FUNCTION_BLOCK FB_Sequence IMPLEMENTS I_Sequence
VAR_INPUT
END_VAR
VAR_OUTPUT
	nNumber:				INT;
END_VAR
VAR
	bStarted:				Bool;
END_VAR

// Quite a lot to do here :-(

METHOD PUBLIC M_Await 
VAR_INPUT
	Message:				STRING(255);
	tTimeout:				TIME;
	bCondition:				BOOL;
	nNumber:				INT;
END_VAR
IF bStarted THEN
	IF bCondition THEN
		THIS^.nNumber:= nNumber;
	END_IF
END_IF
END_METHOD

METHOD M_Reset : BOOL
M_Stop();
nNumber:= -32768;
END_METHOD

METHOD M_Start
bStarted:= TRUE;
END_METHOD

METHOD M_Stop : BOOL
bStarted:= FALSE;
END_METHOD

PROPERTY PUBLIC P_Number : int
GET
P_Number:= nNumber;
END_GET
SET
nNumber:= P_Number;
END_SET
END_PROPERTY

END_FUNCTION_BLOCK

(* stored: Version 1.1.0.1
   POU FB_Sequence: Id {4b1aa270-5e63-4fbf-b9b1-b64186ed4cc4}, SpecialFunc None
   Method M_Await: Id {1bc0e82b-8467-4f35-a54e-996600fba2bc}
   Method M_Reset: Id {4501245b-63d2-4732-9d5e-f656a322de01}
   Method M_Start: Id {0e1345c4-a168-46c5-a849-0de1396f742f}
   Method M_Stop: Id {526a68ea-0096-402e-9748-077658579eca}
   Property P_Number: Id {3cc751bf-6092-4aa8-8de5-3276200b64ad}
   Get Get: Id {92b3a1f5-52d3-44fe-8629-e1295a1ef489}
   Set Set: Id {741fb181-5541-4ab9-8a33-f87392d513c2} *)
